// TIA Portal V20 export
TYPE "CMInterface_AI"
   STRUCT
      ValueIn { ExternalAccessible := 'False'; ExternalVisible := 'False'; ExternalWritable := 'False'} : Real;
   END_STRUCT;
END_TYPE
